// TIA Portal V18 export
DATA_BLOCK "wwwMain_DB"   // DB11
VERSION : 0.1
// stored: AutoNumber true, DBAccessibleFromOPCUA true, DBAccessibleFromWebserver true, InstanceOfName wwwMain, InstanceOfType FB
"wwwMain"
BEGIN
END_DATA_BLOCK
